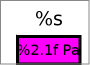
VISUALIZATION Obj_DP_Field  // 90x65
VAR_IN
	rPressValue : REAL;
	sIndex : STRING;
	bPressLimitAlarm : BOOL;
	bPressFailed : BOOL;
	bPressOffline : BOOL;
	bPressExcluded : BOOL;
END_VAR

VAR_IN_OUT
	bSetPressExcluded : BOOL;
	bSetPressIncluded : BOOL;
END_VAR
    Rectangle (16,35 65x30), "%2.1f Pa", text variable: rPressValue, colour toggle: bPressLimitAlarm
    Rectangle (8,4 82x30), "%s", text variable: sIndex
    Rectangle (16,35 65x30), "%2.1f Pa", text variable: rPressValue, invisible if: not bPressExcluded
    Rectangle (16,35 65x30), "OoR", text variable: rPressValue, invisible if: NOT bPressFailed
    Line (80,64) (16,35), invisible if: not bPressExcluded
    Rectangle (16,35 65x30)
        OnMouseClick: OpenDialog Dialog=Dialog_DP_Field, Parameters={bSetPressExcluded: bSetPressExcluded, bSetPressIncluded: bSetPressIncluded, sHeader: sIndex}, Selected={0: , 1: }, OpenModal=True, OpenCentered=True
    Rectangle (16,35 65x30), "%2.1f Pa", text variable: rPressValue, invisible if: not bPressOffline
END_VISUALIZATION

(* stored: Version 1.1.0.1, ProductVersion 3.1.4024.12
   Visu Obj_DP_Field: Id {9f24362b-9e4c-486a-bd75-7f5a57a0dfc2} *)
